// Mitsubishi GX Works2 project: Dodatni poeni   PLC: FX3S
// Dodatni

// task Task_01 (event TRUE, interval 0, priority 31): POU_01

PROGRAM POU_01
VAR
  miks_tecnosti_1 : miks_tecnosti;
  start_but : BOOL;
  stop_but : BOOL;
  ventilcic1 : BOOL;
  ventilcic2 : BOOL;
  ventilcic3 : BOOL;
  motorcic : BOOL;
  senzor11 : BOOL;
  senzor22 : BOOL;
END_VAR
(* structured ladder/FBD written out as ST: instructions are called as NAME(EN, inputs, outputs); _pN, _eN, _tN stand for wires *)
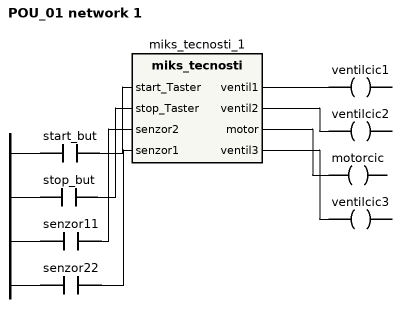
(* network 1 *)
miks_tecnosti_1(start_Taster := start_but, stop_Taster := stop_but, senzor2 := senzor11, senzor1 := senzor22);
ventilcic1 := miks_tecnosti_1.ventil1;
ventilcic2 := miks_tecnosti_1.ventil2;
motorcic := miks_tecnosti_1.motor;
ventilcic3 := miks_tecnosti_1.ventil3;
END_PROGRAM

FUNCTION_BLOCK miks_tecnosti
VAR_INPUT
  start_Taster : BOOL;
  stop_Taster : BOOL;
END_VAR
VAR
  upaljen_sistem : BOOL;
END_VAR
VAR_INPUT
  senzor2 : BOOL;
  senzor1 : BOOL;
END_VAR
VAR_OUTPUT
  ventil1 : BOOL;
  ventil2 : BOOL;
  motor : BOOL;
END_VAR
VAR
  TOF_1 : TOF;
  tajmer_miks_1 : BOOL;
  vrednost_tajmer_miks1 : TIME;
  TOF_2 : TOF;
  TOF_3 : TOF;
  tajmer_miks_2 : BOOL;
  vrednost_tajmer_miks2 : TIME;
  interni : BOOL;
  interni2 : BOOL;
END_VAR
VAR_OUTPUT
  ventil3 : BOOL;
END_VAR
VAR
  interni3 : BOOL;
END_VAR
(* structured ladder/FBD written out as ST: instructions are called as NAME(EN, inputs, outputs); _pN, _eN, _tN stand for wires *)
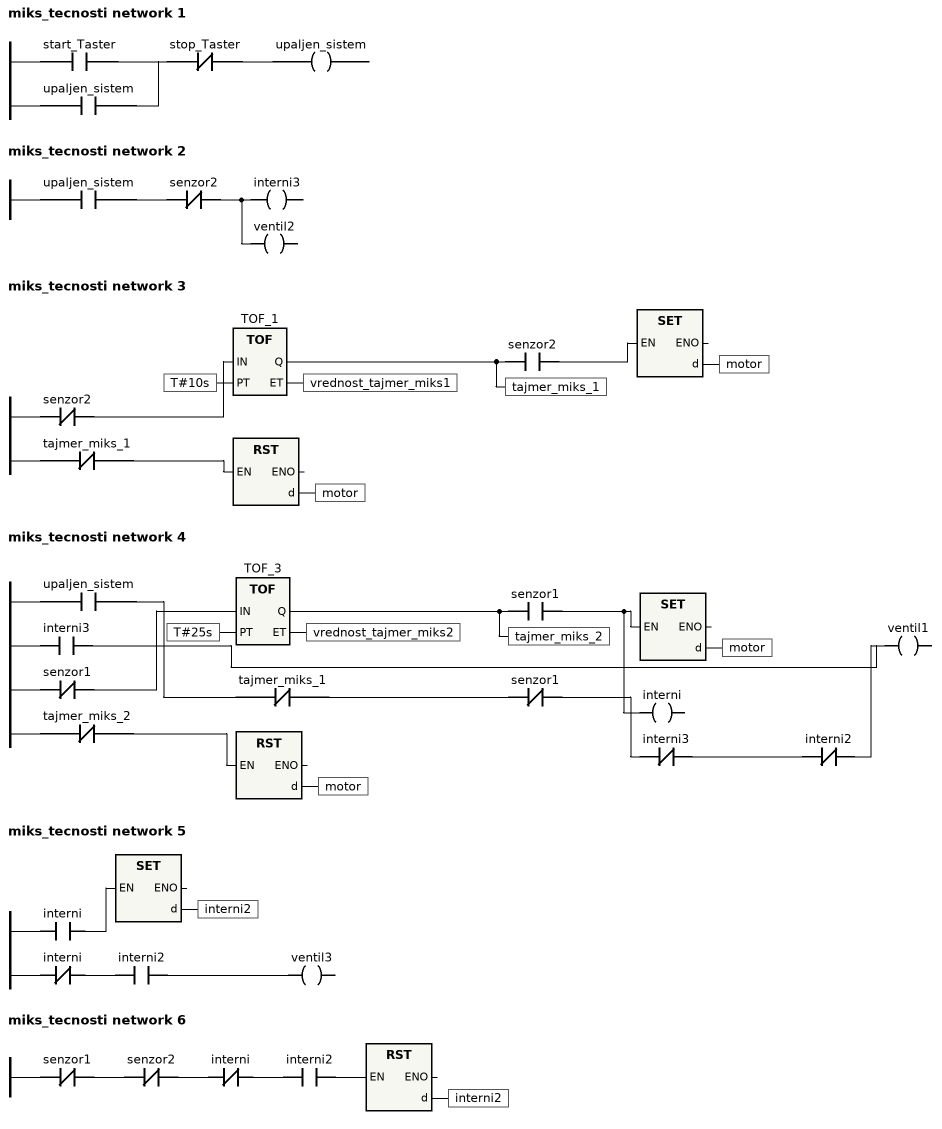
(* network 1 *)
upaljen_sistem := (start_Taster OR upaljen_sistem) AND NOT stop_Taster;
(* network 2 *)
_p1 := upaljen_sistem AND NOT senzor2;
interni3 := _p1;
ventil2 := _p1;
(* network 3 *)
TOF_1(IN := NOT senzor2, PT := T#10s, ET => vrednost_tajmer_miks1);
tajmer_miks_1 := TOF_1.Q;
SET(TOF_1.Q AND senzor2, motor);
RST(NOT tajmer_miks_1, motor);
(* network 4 *)
ventil1 := (upaljen_sistem AND NOT tajmer_miks_1 AND NOT senzor1 AND NOT interni3 AND NOT interni2) OR interni3;
TOF_3(IN := NOT senzor1, PT := T#25s, ET => vrednost_tajmer_miks2);
_p1 := TOF_3.Q AND senzor1;
interni := _p1;
SET(_p1, motor);
tajmer_miks_2 := TOF_3.Q;
RST(NOT tajmer_miks_2, motor);
(* network 5 *)
SET(interni, interni2);
ventil3 := NOT interni AND interni2;
(* network 6 *)
RST(NOT senzor1 AND NOT senzor2 AND NOT interni AND interni2, interni2);
END_FUNCTION_BLOCK
